PROGRAM MAIN
VAR
	(* *) (* *) (* *) (* *) (* *) (* *) (* *) (* *) (* *) (* *) (* *) (* *) (* *)
	meter1: LREAL;
	meter2: LREAL;	
	meter3: LREAL;	
	meter4: LREAL;	
	meter5: LREAL;	
	(* *) (* *) (* *) (* *) (* *) (* *) (* *) (* *) (* *) (* *) (* *) (* *) (* *)
	idx: BOOL;
	idxDev: BOOL;
	(* *) (* *) (* *) (* *) (* *) (* *) (* *) (* *) (* *) (* *) (* *) (* *) (* *)
END_VAR
VAR
END_VAR

(*
start item = [] consist of fx1,fx2,fx3,fx4,fx5 and are assigned to output terminals 
meter = [] sample consists of metrics conversions from LREAL TO INT and loses some information
io.pX_REF = [] sample commandsio.p1_REF,io.p2_REF,io.p3_REF,io.p4_REF,io.p5_REF vars interconnected to ->
IF -loop where when assigned True enables IO variable write to io.k1_REF,io.k2_REF,io.k3_REF,io.k4_REF,io.k5_REF
in which assigned vars are INTs and enable to control flow directly from the terminal output to item input. 
*)
(* *) (* *) (* *) (* *) (* *) (* *) (* *) (* *) (* *) (* *) (* *) (* *) (* *)
(* *) (* *) (* *) (* *) (* *) (* *) (* *) (* *) (* *) (* *) (* *) (* *) (* *)
(* *) (* *) (* *) (* *) (* *) (* *) (* *) (* *) (* *) (* *) (* *) (* *) (* *)
(* *) (* *) (* *) (* *) (* *) (* *) (* *) (* *) (* *) (* *) (* *) (* *) (* *)
(* *) (* *) (* *) (* *) (* *) (* *) (* *) (* *) (* *) (* *) (* *) (* *) (* *)
(* *) (* *) (* *) (* *) (* *) (* *) (* *) (* *) (* *) (* *) (* *) (* *) (* *)
(* *) (* *) (* *) (* *) (* *) (* *) (* *) (* *) (* *) (* *) (* *) (* *) (* *)
(* *) (* *) (* *) (* *) (* *) (* *) (* *) (* *) (* *) (* *) (* *) (* *) (* *)
(* *) (* *) (* *) (* *) (* *) (* *) (* *) (* *) (* *) (* *) (* *) (* *) (* *)
(* *) (* *) (* *) (* *) (* CURRENT CONTROL *) (* *) (* *) (* *) (* *) (* *)
IF IO.p1_REF = TRUE THEN
	IO.k1_REF:=10000;
	ELSE
		IO.k1_REF:=0;	
END_IF
(* *) (* *) (* *) (* *) (* VOLTAGE CONTROL *) (* *) (* *) (* *) (* *) (* *)
IF IO.p2_REF = TRUE THEN
	IO.k2_REF:=10000;
	ELSE
		IO.k2_REF:=0;	
END_IF
(* *) (* *) (* *) (* *) (* VOLTAGE CONTROL *) (* *) (* *) (* *) (* *) (* *)
IF IO.p3_REF = TRUE THEN
	IO.k3_REF:=10000;
	ELSE
		IO.k3_REF:=0;	
END_IF
(* *) (* *) (* *) (* *) (* VOLTAGE CONTROL *) (* *) (* *) (* *) (* *) (* *)
IF IO.p4_REF = TRUE THEN
	IO.k4_REF:=10000;
	ELSE
		IO.k4_REF:=0;	
END_IF
(* *) (* *) (* *) (* *) (* VOLTAGE CONTROL *) (* *) (* *) (* *) (* *) (* *)
IF IO.p5_REF = TRUE THEN
	IO.k5_REF:=10000;
	ELSE
		IO.k5_REF:=0;	
END_IF
(* *) (* *) (* *) (* *) (* *) (* *) (* *) (* *) (* *) (* *) (* *) (* *) (* *)
(* *) (* *) (* *) (* *) (* *) (* *) (* *) (* *) (* *) (* *) (* *) (* *) (* *)
(* *) (* *) (* *) (* *) (* *) (* *) (* *) (* *) (* *) (* *) (* *) (* *) (* *)
(* *) (* *) (* *) (* *) (* *) (* *) (* *) (* *) (* *) (* *) (* *) (* *) (* *)
(* *) (* *) (* *) (* *) (* *) (* *) (* *) (* *) (* *) (* *) (* *) (* *) (* *)
(* *) (* *) (* *) (* *) (* *) (* *) (* *) (* *) (* *) (* *) (* *) (* *) (* *)
(* *) (* *) (* *) (* *) (* *) (* *) (* *) (* *) (* *) (* *) (* *) (* *) (* *)
(* *) (* *) (* *) (* *) (* *) (* *) (* *) (* *) (* *) (* *) (* *) (* *) (* *)
IF IO.p1_REF = TRUE THEN
	IO.k1_REF:=10000;
	ELSE
		IO.k1_REF:=0;	
END_IF
(* *) (* *) (* *) (* *) (* *) (* *) (* *) (* *) (* *) (* *) (* *) (* *) (* *)
(* *) (* *) (* *) (* *) (* *) (* *) (* *) (* *) (* *) (* *) (* *) (* *) (* *)
(* *) (* *) (* *) (* *) (* *) (* *) (* *) (* *) (* *) (* *) (* *) (* *) (* *)
(* *) (* *) (* *) (* *) (* *) (* *) (* *) (* *) (* *) (* *) (* *) (* *) (* *)
(* *) (* *) (* *) (* *) (* CLOSES ALL VALVES *) (* *) (* *) (* *) (* *) (* *)
IF IO.erikoismuuttujaSum=TRUE OR io.r1_REF =TRUE AND io.r2_REF =TRUE AND io.r3_REF =TRUE AND io.r4_REF =TRUE AND io.r5_REF =TRUE AND io.r6_REF =TRUE AND io.v1_REF =TRUE AND io.v2_REF =TRUE AND idx =TRUE THEN
		idx:=TRUE;
	io.r1_REF:=TRUE;
	io.r2_REF:=TRUE;	
			io.r3_REF:=TRUE;
	io.r4_REF:=TRUE;
			io.r5_REF:=TRUE;
	io.r6_REF:=TRUE;
			io.v1_REF:=TRUE;
	io.v2_REF:=TRUE;
	END_IF
(* *) (* *) (* *) (* *) (* *) (* *) (* *) (* *) (* *) (* *) (* *) (* *) (* *)
(* *) (* *) (* *) (* *) (* *) (* *) (* *) (* *) (* *) (* *) (* *) (* *) (* *)
(* *) (* *) (* *) (* *) (* *) (* *) (* *) (* *) (* *) (* *) (* *) (* *) (* *)
(* *) (* *) (* *) (* *) (* *) (* *) (* *) (* *) (* *) (* *) (* *) (* *) (* *)
(* *) (* *) (* *) (* *) (* KEEPS VALVES CLOSED *) (* *) (* *) (* *) (* *) (* *)
IF IO.erikoismuuttujaSum=FALSE AND idx=TRUE THEN
	idx:=FALSE;
			io.r1_REF:=FALSE;
	io.r2_REF:=FALSE;
			io.r3_REF:=FALSE;
	io.r4_REF:=FALSE;
			io.r5_REF:=FALSE;
	io.r6_REF:=FALSE;
			io.v1_REF:=FALSE;
	io.v2_REF:=FALSE;
END_IF
(* *) (* *) (* *) (* *) (* *) (* *) (* *) (* *) (* *) (* *) (* *) (* *) (* *)
///////////////////////////////////////////////////////////////////////////
(* *) (* *) (* *) (* *) (* *) (* *) (* *) (* *) (* *) (* *) (* *) (* *) (* *)
///////////////////////////////////////////////////////////////////////////
(* *) (* *) (* *) (* *) (* *) (* *) (* *) (* *) (* *) (* *) (* *) (* *) (* *)
(*CONVERTS LREAL ITEM OUTPUTS INTO TERMINAL INPUTS OF INT OF REAL WORLD SCALE*)
meter1:=io.f1_REF/520 (*25 ml/min*) (*/819.5*100*); //ADD CONVERSION // AGD ? CURRENT
meter2:=io.f2_REF/520 (*25 ml/min*) (*/819.5*100*); //ADD CONVERSION // VOLTAGE
meter3:=io.f3_REF/520 (*25 ml/min*) (*/819.5*100*); //ADD CONVERSION // VOLTAGE
meter4:=io.f4_REF/520 (*25 ml/min*) (*/819.5*100*); //ADD CONVERSION // VOLTAGE
meter5:=io.f5_REF/520 (*25 ml/min*) (*/819.5*100*); //ADD CONVERSION // VOLTAGE
// k1_REF AS OVERRIDING ODD INPUT VALUES
// 
// meter1:=io.k1_REF/31 (* N ml/min *) (*/819.5*100*); //ADD CONVERSION // AGD ? CURRENT
// meter2:=io.k2_REF/31 (* N ml/min *) (*/819.5*100*); //ADD CONVERSION // VOLTAGE
// meter3:=io.k3_REF/31 (* N ml/min *) (*/819.5*100*); //ADD CONVERSION // VOLTAGE
// meter4:=io.k4_REF/31 (* N ml/min *) (*/819.5*100*); //ADD CONVERSION // VOLTAGE
// meter5:=io.k5_REF/31 (* N ml/min *) (*/819.5*100*); //ADD CONVERSION // VOLTAGE
//  
(* *) (* *) (* *) (* *) (* *) (* *) (* *) (* *) (* *) (* *) (* *) (* *) (* *)
(* *) (* *) (* *) (* *) (* *) (* *) (* *) (* *) (* *) (* *) (* *) (* *) (* *)
(* *) (* *) (* *) (* *) (* *) (* *) (* *) (* *) (* *) (* *) (* *) (* *) (* *)
(* *) (* *) (* *) (* *) (* *) (* *) (* *) (* *) (* *) (* *) (* *) (* *) (* *)
(* *) (* *) (* *) (* *) (* *) (* *) (* *) (* *) (* *) (* *) (* *) (* *) (* *)
(* *) (* *) (* *) (* *) (* *) (* *) (* *) (* *) (* *) (* *) (* *) (* *) (* *)
(* *) (* *) (* *) (* *) (* *) (* *) (* *) (* *) (* *) (* *) (* *) (* *) (* *)
(* *) (* *) (* *) (* *) (* *) (* *) (* *) (* *) (* *) (* *) (* *) (* *) (* *)
(* *) (* *) (* *) (* *) (* *) (* *) (* *) (* *) (* *) (* *) (* *) (* *) (* *)
(* *) (* *) (* *) (* *) (* *) (* *) (* *) (* *) (* *) (* *) (* *) (* *) (* *)
(* *) (* *) (* *) (* *) (* *) (* *) (* *) (* *) (* *) (* *) (* *) (* *) (* *)
(* *) (* *) (* *) (* *) (* *) (* *) (* *) (* *) (* *) (* *) (* *) (* *) (* *)

END_PROGRAM

(* stored: Version 1.1.0.1, ProductVersion 3.1.4024.0
   POU MAIN: Id {9073a552-bc51-47bc-a064-e3f15f7ee309}, SpecialFunc None *)
